DATA_BLOCK "Hebeanlage_DB_1"
{ S7_Optimized_Access := 'TRUE' }
VERSION : 0.1
NON_RETAIN
"Hebeanlage"

BEGIN

END_DATA_BLOCK

